ABB RobotStudio station: 码垛.rspag

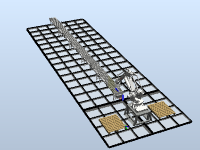
--- station ---
Station PartC (saved by RobotStudio 6.8.8148.134)
Controller System1, task T_ROB1: task frame (RAPID world) sits at (-2000, 0, 800) mm in the station
Controller System1
  mechanical unit ROB_1: IRB660_180_315__01, 6 joints, base frame (0, 0, 0) mm
Layout (positions relative to the parent item):
  - 部件_2 [part] at (0, 0, 23.06) mm
  - ChuanSongDai [smart component]
      signals: DO jiance, DO daowei
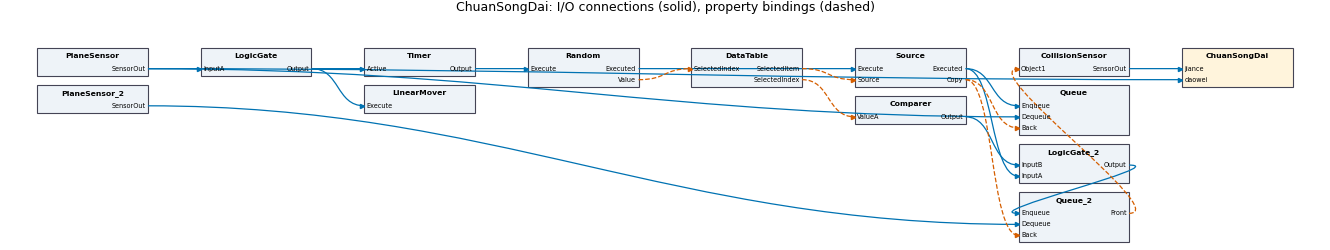
      connections:
        Timer.Output -> Random.Execute
        Random.Executed -> Source.Execute
        LogicGate.Output -> LinearMover.Execute
        Source.Executed -> Queue.Enqueue
        PlaneSensor.SensorOut -> Queue.Dequeue
        LogicGate.Output -> Timer.Active
        Comparer.Output -> LogicGate_2.InputB
        Source.Executed -> LogicGate_2.InputA
        PlaneSensor.SensorOut -> LogicGate.InputA
        LogicGate_2.Output -> Queue_2.Enqueue
        PlaneSensor_2.SensorOut -> Queue_2.Dequeue
        CollisionSensor.SensorOut -> ChuanSongDai.jiance
        PlaneSensor.SensorOut -> ChuanSongDai.daowei
        Random.Value => DataTable.SelectedIndex
        DataTable.SelectedItem => Source.Source
        Source.Copy => Queue.Back
        DataTable.SelectedIndex => Comparer.ValueA
        Source.Copy => Queue_2.Back
        Queue_2.Front => CollisionSensor.Object1
    - Timer [smart component, from Components\Timer.rslib]
        properties: StartTime=0.1; Interval=2.1; Repeat=true; CurrentTime=65.88
    - Random [smart component, from Components\Random.rslib]
        properties: Value=0.822097293018409; Min=0; Max=1
    - DataTable [smart component, from Components\DataTable.rslib]
        properties: DataType=Object; NumItems=2; SelectedIndex=1; SelectedItem=绿; Item0=红; Item1=绿
    - Source [smart component, from Components\Source.rslib]
        properties: Source=绿; Copy=(none); Parent=(none); Position=[12.3 0.05 0.8]; Orientation=[0 0 0]; Transient=false; PhysicsBehavior=0
    - Queue [smart component, from Components\Queue.rslib]
        properties: Back=(none); Front=(none); Queue={f225a319-0da6-49b0-b8ed-6a01384f5e4a};{a5013529-57de-4880-b6b7-02fcb26c5601};{ef2480c9-5506-4bd8-9223-d6bf2a21d1ab};{0e0a0a7f-5876-4dd6-bb12-e12ef663cda4};{136b776b-8417-404b-a9ca-a707fcf896fa};{cb7463a0-53d0-4ea9-9850-c55b52504a23};{429f5040-d4eb-4fed-af85-08b79dd3797b};{eae50fed-bce9-4253-838e-1ef2825aae45};{02ee2a03-807e-4b62-b245-e530b87cc1ef};{56b14a6d-97e9-4dc3-87d2-51b8ae3edd15};{4860391a-c953-42ac-88c5-ff0e025b596f};{e91e6b01-9356-4c41-92bb-629052fa1d8e};{204cb33b-3ecf-4ce5-996c-fe7c59920a57};{7c8b56eb-ca14-4c06-a856-6019091091a4};{df6cc59b-68ab-44d0-93b8-b393a520ffed};{0df2fced-d373-4a8c-8570-b0d5d7a52f36};{2e525211-6f58-4c05-9e0c-770fe7f0b080};{2d23c5ff-243a-4a38-8aa8-df9699042488};{c13a5a0e-5a8c-4728-abd8-7e4e8a2dcb0f};{516486e3-0f15-4dc5-a66e-dbea303b17aa};{aaca48b5-e3d4-4e57-b6f3-5a542b0a9696};{807b33c7-9c87-478a-ab71-3c40786a7147};{5f0bf4f3-3df5-4e69-bf08-9b9bc90daa45};{4c77b5d5-784e-45a8-9efe-70001206c053};{c7fe08fd-9e7d-46e3-a402-e1c13f8510d7};{9c7207f7-ca42-4ffb-ba10-967dca55547d};{a7cd077e-332a-445c-8b65-e16c12a6adc8};{2053ef60-9d1c-42bc-a075-6101035489ef};{a5b924c0-e777-4755-b462-75c4f45590d4};{88fdcb66-1964-4a9a-9fd3-ca14f0fdc147};{ef60cde5-ce41-4944-b10e-df7ae6d2f20b};{427c14b4-609a-4b20-a2be-5ba79a59d804};{fb550f5b-ebcd-4dd1-8fa9-009c54dba658};{c15f4878-baa5-4e14-8903-3b1b5c857eef};{6ededeb0-61e9-45d7-b110-e43846e68698};{d93d9120-f688-4177-bbd5-c04ba3deb883};{aed52de2-8a50-4a30-962b-f942badb32ba};{0d4db61c-ee27-4f7b-9537-b14f67708c8e};{f394902b-ba95-4894-9040-dd871542cf1b};{d8c25479-f3b6-4551-bfd2-063a150a2d78};{38238fd8-de79-4013-ad54-694b5345ed3f};{5bd13c71-3d62-4c6d-bbbc-cc516422125c};{07b92203-4d3e-45b5-80a9-1ec55a767f10};{a74c1ad0-5c37-4e0d-81f5-31d5f0e208c7};{758074db-41a4-4db3-98d0-906284b01602};{6d04588b-afa6-4a99-82e4-be17e8210f91};{348561f2-af5d-4f36-8eda-e8a6df29ee32};{b923b243-db1b-4daf-bb9b-77d6146748ea};{a27ccf1c-a8f2-4afc-910f-c603e908e337};{821874ad-1724-42f4-bffa-9c6221594dbd};{ef4ad952-7e1f-4f76-99cc-78a6cae096f3};{1f82013b-60b1-4451-ab71-6434a119db9b};{6f134922-b885-41ab-a43e-bbaa37394d8e};{7190a3ba-ed00-41fa-baa9-cd3fce09d1b0};{2d9f646b-25f1-493c-9c88-1cc082209cb0};{1953191b-e8a9-4a7b-8072-886da8d2683f};{e6bacfb4-f14c-4f22-ab39-c3f0abe42d56};{8f446c08-29c5-4440-b72c-75c0776f3732};{2ac58cdd-d2f5-4fc3-992e-0072fed280bc};{aa8b40f0-69ac-4ba4-a17b-86b932449b98};{9f18385d-f857-4cee-ba85-427a449adb07};{50a51e2c-eaa8-4e6c-b4d6-fb4141048cc5};{d0e21a90-9519-43be-867c-222b4f1f38a1};{7b820672-940c-4b0d-92fa-2fe77afa0e85};{c9ad62ae-d9f6-4551-810e-0b3d00224a97};{c4bdeaf5-84be-4565-9116-5f2757d6e74e};{59238313-e22c-43d2-a97a-5d6b7997641f};{2edab753-53a4-48c2-8791-8efd26fc352b};{26800b2b-b13d-4846-b0fd-fb68af482c4b};{f6f03289-8baf-42de-9ffb-846ca9933dae};{1e187082-cda8-4acf-9a05-f0e611de5223};{185980c2-df0e-4768-98ff-8c0ecfa9ede1};{c493306c-ebd5-48b7-94e6-332e50b6f699};{c7ce4e63-1a53-4056-bb2e-8373dea2df1b};{00ae25b9-8afd-4489-9d6e-e100ffd902fb};{a46d434a-4951-431b-bf92-58fad4eae258};{0ac38f34-9f27-4a73-b789-8751a30c78c9};{415bd256-8ea2-40f1-afb7-912d3eb54ad5};{5b8083c6-e57c-4f6b-b63b-b57aa365888c};{33a629bd-e383-481d-ba6f-0150e17603ca};{c31adef7-9013-47b8-8c02-a895f65a4230};{bc88b68d-7d5b-4bfa-85ac-205ac4b92c3f};{d122ac05-f8f7-4393-bed0-9e9b9361324e};{227dc145-5e4e-4412-a5e8-4d724cccd912};{96275f03-4ecc-469c-b843-ec3ce2da747c};{3a609a9e-e66e-4842-80c6-6da2b92c4aab};{36be5265-f703-4688-b700-c963585c6167};{78c7701e-fa20-47d5-ad67-3c0217d249c5};{4e3675bd-98e1-4d49-9126-e21ce655e718};{d18456cf-9ef5-48aa-9364-d375af649ce2};{b12914ea-076e-4431-85c1-3df9dfa51120};{477bcbfa-4fa5-46f0-968d-82c75168f6dd};{06c00f79-e598-488f-ab9b-14e942d20a45};{fa9f11b3-aab2-4e3c-9f67-386e2b048710};{965c1e25-d47d-434e-af53-90d46d55ac75};{4f6779af-fb5c-4c41-8ac5-645e945892b7};{961cba95-9dcf-4a6f-ae69-a71c8ac9bd9b};{c1c4ceb7-0aac-4022-8558-a4c71beaa21c};{0f13d351-420a-472e-9a7e-8c0a797d1716};{805a9eb2-f81c-40c7-8f83-e398ffb0342c}; NumberOfObjects=7
    - 600_guide [part, from Equipment\Conveyor Guide 600.rslib]
    - LinearMover [smart component, from Components\LinearMover.rslib]
        properties: Object=Queue; Direction=[-0.001 0 0]; Speed=0.8; Reference=Global; ReferenceObject=(none)
    - PlaneSensor [smart component, from Components\PlaneSensor.rslib]
        properties: Origin=[0 0 0.8]; Axis1=[0 0.6 0]; Axis2=[0 0.1 0.15]; SensedPart=(none)
      - _sensorPart_ [part]
    - LogicGate [smart component, from Components\LogicGate.rslib]
        properties: Operator=NOT; Delay=0
    - Comparer [smart component, from Components\Comparer.rslib]
        properties: ValueA=1; Operator===; ValueB=0
    - LogicGate_2 [smart component, from Components\LogicGate.rslib]
        properties: Operator=AND; Delay=0
    - Queue_2 [smart component, from Components\Queue.rslib]
        properties: Back=(none); Front=(none); Queue={f72ca3a7-ed19-412f-a648-57eb43a8f19a};{0d191394-6de3-422a-92fa-47054eac63d5};{95f6c7dd-c1c0-4261-85cb-418d534c64aa};{209a704b-017e-4eed-926c-5e79c4908886};{0d8d839c-5b7f-48c1-871d-9d79d5e8a973};{1d3bda1c-354e-4164-852e-5573aebfca0e};{d40879a3-4785-47c6-84ec-f61648f74983};{a7cc7dfc-d99a-413b-9ad3-ab5f673166e2};{438c7bca-c9a8-4b7b-9a0a-5120735f9a42};{f225a319-0da6-49b0-b8ed-6a01384f5e4a};{0e0a0a7f-5876-4dd6-bb12-e12ef663cda4};{136b776b-8417-404b-a9ca-a707fcf896fa};{cb7463a0-53d0-4ea9-9850-c55b52504a23};{429f5040-d4eb-4fed-af85-08b79dd3797b};{7c8b56eb-ca14-4c06-a856-6019091091a4};{0df2fced-d373-4a8c-8570-b0d5d7a52f36};{516486e3-0f15-4dc5-a66e-dbea303b17aa};{aaca48b5-e3d4-4e57-b6f3-5a542b0a9696};{5f0bf4f3-3df5-4e69-bf08-9b9bc90daa45};{4c77b5d5-784e-45a8-9efe-70001206c053};{c7fe08fd-9e7d-46e3-a402-e1c13f8510d7};{9c7207f7-ca42-4ffb-ba10-967dca55547d};{88fdcb66-1964-4a9a-9fd3-ca14f0fdc147};{ef60cde5-ce41-4944-b10e-df7ae6d2f20b};{fb550f5b-ebcd-4dd1-8fa9-009c54dba658};{6ededeb0-61e9-45d7-b110-e43846e68698};{758074db-41a4-4db3-98d0-906284b01602};{6d04588b-afa6-4a99-82e4-be17e8210f91};{348561f2-af5d-4f36-8eda-e8a6df29ee32};{b923b243-db1b-4daf-bb9b-77d6146748ea};{6f134922-b885-41ab-a43e-bbaa37394d8e};{1953191b-e8a9-4a7b-8072-886da8d2683f};{e6bacfb4-f14c-4f22-ab39-c3f0abe42d56};{2ac58cdd-d2f5-4fc3-992e-0072fed280bc};{aa8b40f0-69ac-4ba4-a17b-86b932449b98};{9f18385d-f857-4cee-ba85-427a449adb07};{d0e21a90-9519-43be-867c-222b4f1f38a1};{c9ad62ae-d9f6-4551-810e-0b3d00224a97};{c4bdeaf5-84be-4565-9116-5f2757d6e74e};{2edab753-53a4-48c2-8791-8efd26fc352b};{26800b2b-b13d-4846-b0fd-fb68af482c4b};{1e187082-cda8-4acf-9a05-f0e611de5223};{00ae25b9-8afd-4489-9d6e-e100ffd902fb};{a46d434a-4951-431b-bf92-58fad4eae258};{5b8083c6-e57c-4f6b-b63b-b57aa365888c};{33a629bd-e383-481d-ba6f-0150e17603ca};{c31adef7-9013-47b8-8c02-a895f65a4230};{3a609a9e-e66e-4842-80c6-6da2b92c4aab};{36be5265-f703-4688-b700-c963585c6167};{d18456cf-9ef5-48aa-9364-d375af649ce2};{b12914ea-076e-4431-85c1-3df9dfa51120};{fa9f11b3-aab2-4e3c-9f67-386e2b048710};{965c1e25-d47d-434e-af53-90d46d55ac75};{4f6779af-fb5c-4c41-8ac5-645e945892b7};{961cba95-9dcf-4a6f-ae69-a71c8ac9bd9b}; NumberOfObjects=4
    - CollisionSensor [smart component, from Components\CollisionSensor.rslib]
        properties: Object1=(none); Object2=检测; NearMiss=0; Part1=(none); Part2=(none); CollisionType=0
    - PlaneSensor_2 [smart component, from Components\PlaneSensor.rslib]
        properties: Origin=[0 0.7 0.77]; Axis1=[1 0 0]; Axis2=[0 0 1]; SensedPart=(none)
      - _sensorPart_ [part]
  - 红 [part] at (2300, 50, 800) mm
  - 绿 [part]
  - 检测 [part] at (20, 0, 0) mm
  - DiZuo [part] at (-2000, 0, 800) mm
  - IRB660_180_315__01 [mechanism, from Robots\IRB660_180_315__01.rslib] at (-2000, 0, 800) mm; joint values [0.1259, 0.727, 0.7593, 0.1259] (rad or m)
  - TuoPan_Left [part, from B站\木托.rslib] at (-2900, 1230, 0) mm, rotated rx 90 ry 0 rz 90 deg
  - TuoPan_Right [part, from B站\木托.rslib] at (-2900, -2460, 0) mm, rotated rx 90 ry 0 rz 90 deg
  - XiPan [smart component]
      signals: DI zhuaqu
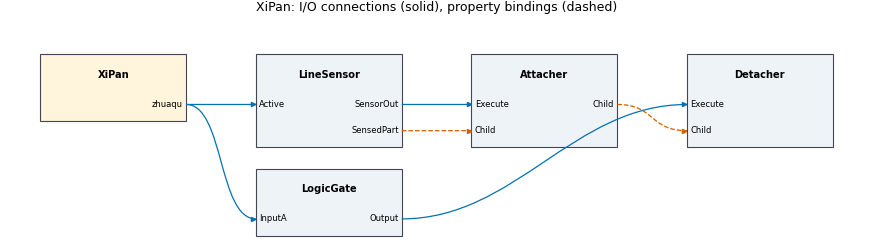
      connections:
        LineSensor.SensorOut -> Attacher.Execute
        LogicGate.Output -> Detacher.Execute
        XiPan.zhuaqu -> LineSensor.Active
        XiPan.zhuaqu -> LogicGate.InputA
        LineSensor.SensedPart => Attacher.Child
        Attacher.Child => Detacher.Child
    - Attacher [smart component, from Components\Attacher.rslib]
        properties: Parent=MyTool; Flange=0; Child=(none); Mount=false; Offset=[0 0 0]; Orientation=[0 0 0]
    - Detacher [smart component, from Components\Detacher.rslib]
        properties: Child=(none); KeepPosition=true
    - LineSensor [smart component, from Components\LineSensor.rslib] at (371, 300, 1200) mm, rotated rx 180 ry 0 rz -180 deg
        properties: Start=[3.44022367537722E-07 -3.10121215152392E-07 -0.0200000204160531]; End=[3.44022367537722E-07 -3.10121215152392E-07 0.029999979583947]; Radius=0.003; SensedPart=(none); SensedPoint=[-1.62997448730469 -2.08514575195312 1.35087182617188]
      - _sensorPart_ [part]
    - MyTool [mechanism] at (371, 300, 1380) mm, rotated rx 180 ry 0 rz -180 deg
        TCP MyTool at (0, 0, 180) mm
        links: 吸盘夹具600_400.
    - LogicGate [smart component, from Components\LogicGate.rslib]
        properties: Operator=NOT; Delay=0
  - 600_guide [part, from Equipment\Conveyor Guide 600.rslib] at (3000, 0, 0) mm
  - 600_guide_2 [part, from Equipment\Conveyor Guide 600.rslib] at (6000, 0, 0) mm
  - 600_guide_3 [part, from Equipment\Conveyor Guide 600.rslib] at (9000, 0, 0) mm
  - 600_guide_4 [part, from Equipment\Conveyor Guide 600.rslib] at (12000, 0, 0) mm
Attachment: LineSensor is attached to MyTool / 吸盘夹具600_400.
Attachment: MyTool is attached to IRB660_180_315__01 / Link6
EventTableEntry 2443: Group=, Trigger=DO_007 2444, Actions=[EventTableActionMechanicalPose 2445], Comment=, ActivationMode=2, Cyclic=false
EventTableTriggerIO 2444: IOValue=[1], IRC5Controller=? -1, Operator=0, SignalSource=? -1
EventTableActionMechanicalPose 2445: VirtualSignal=, Mechanism=? -1, ToPoseName=SyncPosition, VirtualSignalValue=[1]
EventTableEntry 2446: Group=, Trigger=DO_007 2447, Actions=[EventTableActionMechanicalPose 2448], Comment=, ActivationMode=2, Cyclic=false
EventTableTriggerIO 2447: IOValue=[0], IRC5Controller=? -1, Operator=0, SignalSource=? -1
EventTableActionMechanicalPose 2448: VirtualSignal=, Mechanism=? -1, ToPoseName=HomePosition, VirtualSignalValue=[1]
Station logic (signal -> signal, property => property):
  System1.ZhuaQu -> XiPan.zhuaqu
  ChuanSongDai.daowei -> System1.DaoWei
  ChuanSongDai.jiance -> System1.JianCe
Targets, tools, work objects and paths stored in the station and not in the controller backup, written as RAPID:
! task T_ROB1
MODULE CalibData
  PERS tooldata tool1:=[TRUE,[[15.5,0,69.3],[1,0,0,0]],[1,[0,0,1],[1,0,0,0],0,0,0]];
  PERS tooldata tool2:=[TRUE,[[-22.5,0,83.554],[1,0,0,0]],[1,[0,0,1],[1,0,0,0],0,0,0]];
  PERS tooldata tool3:=[TRUE,[[-22.5,0,160.554],[1,0,0,0]],[1,[0,0,1],[1,0,0,0],0,0,0]];
  PERS tooldata Tooldata_4:=[TRUE,[[15.5,0,69.3],[1,0,0,0]],[1,[0,0,1],[1,0,0,0],0,0,0]];
  PERS tooldata Tooldata_5:=[TRUE,[[-22.5,0,83.554],[1,0,0,0]],[1,[0,0,1],[1,0,0,0],0,0,0]];
  PERS tooldata Tooldata_6:=[TRUE,[[-22.5,0,160.554],[1,0,0,0]],[1,[0,0,1],[1,0,0,0],0,0,0]];
ENDMODULE

! task T_ROB1
MODULE Module1
  CONST robtarget Target_10:=[[2810,-1230,2303],[0,0,1,0],[0,0,0,0],[9E+09,9E+09,9E+09,9E+09,9E+09,9E+09]];
ENDMODULE


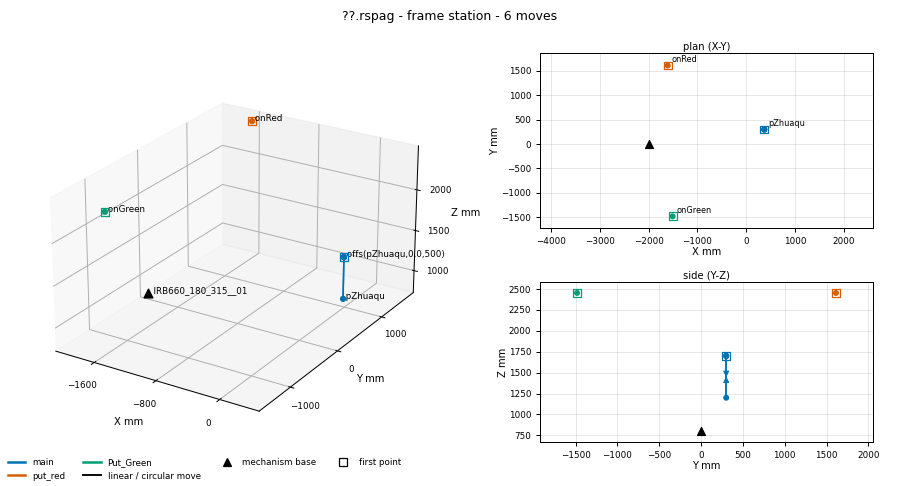
[picture p0: tool path of 码垛.rspag in frame station, 6 of 49 moves have a stored position in this frame; points joined in program order, loops and branches not executed]
--- Backups/System1/RAPID/TASK1/PROGMOD/CalibData.mod ---
MODULE CalibData
	PERS tooldata MyTool:=[TRUE,[[0,0,180],[1,0,0,0]],[1,[0,0,1],[1,0,0,0],0,0,0]];
	TASK PERS wobjdata Work1:=[FALSE,TRUE,"",[[-900,1230,-650],[1,0,0,0]],[[0,0,0],[1,0,0,0]]];
	TASK PERS wobjdata Work2:=[FALSE,TRUE,"",[[620,-1190,-650],[0,0,0,1]],[[0,0,0],[1,0,0,0]]];
ENDMODULE

--- Backups/System1/RAPID/TASK1/PROGMOD/Module1.mod ---
MODULE Module1
	CONST jointtarget Home:=[[0,0,0,0,0,0],[9E+9,9E+9,9E+9,9E+9,9E+9,9E+9]];

	CONST robtarget pZhuaqu:=[[2371.00,300.00,400.00],[1.79568E-6,3.56064E-9,-1,2.27205E-7],[0,0,0,0],[9E+9,9E+9,9E+9,9E+9,9E+9,9E+9]];
	CONST robtarget pFang1:=[[375.00,250.00,400.00],[6.05115E-7,7.10411E-9,1,-1.70585E-6],[1,0,1,0],[9E+9,9E+9,9E+9,9E+9,9E+9,9E+9]];
	CONST robtarget pFang2:=[[1145.00,250.00,400.00],[2.95605E-7,3.17763E-8,-1,1.78569E-6],[0,0,0,0],[9E+9,9E+9,9E+9,9E+9,9E+9,9E+9]];
	CONST robtarget pFang3:=[[250.00,895.00,400.00],[8.4952E-7,0.707106,-0.707107,1.59825E-6],[1,0,0,0],[9E+9,9E+9,9E+9,9E+9,9E+9,9E+9]];
    CONST robtarget pFang4:=[[750.00,895.00,400.00],[8.4952E-7,0.707106,-0.707107,1.59825E-6],[1,0,0,0],[9E+9,9E+9,9E+9,9E+9,9E+9,9E+9]];
	CONST robtarget pFang5:=[[1250.00,895.00,400.00],[8.4952E-7,0.707106,-0.707107,1.59825E-6],[1,0,0,0],[9E+9,9E+9,9E+9,9E+9,9E+9,9E+9]];

    CONST robtarget p2Fang1:=[[250.00,375.00,800.00],[8.4952E-7,0.707106,-0.707107,1.59825E-6],[1,0,0,0],[9E+9,9E+9,9E+9,9E+9,9E+9,9E+9]];
	CONST robtarget p2Fang2:=[[770.00,375.00,800.00],[8.4952E-7,0.707106,-0.707107,1.59825E-6],[1,0,0,0],[9E+9,9E+9,9E+9,9E+9,9E+9,9E+9]];
	CONST robtarget p2Fang3:=[[1250.00,375.00,800.00],[1.27986E-6,-0.707107,-0.707107,-1.27986E-6],[-2,0,0,0],[9E+9,9E+9,9E+9,9E+9,9E+9,9E+9]];
    CONST robtarget p2Fang4:=[[375.00,1020.00,800.00],[6.05115E-7,7.10411E-9,1,-1.70585E-6],[1,0,1,0],[9E+9,9E+9,9E+9,9E+9,9E+9,9E+9]];
    CONST robtarget p2Fang5:=[[1145.00,1020.00,800.00],[6.05115E-7,7.10411E-9,1,-1.70585E-6],[1,0,1,0],[9E+9,9E+9,9E+9,9E+9,9E+9,9E+9]];

    CONST robtarget pPut_green3:=[[250.00,895.00,400.00],[1.03654E-6,0.707107,-0.707107,1.4838E-6],[-1,0,0,0],[9E+9,9E+9,9E+9,9E+9,9E+9,9E+9]];
	CONST robtarget pPut_green1:=[[375.00,250.00,400.00],[1.78435E-6,1,1.03949E-8,3.03588E-7],[-1,0,-1,0],[9E+9,9E+9,9E+9,9E+9,9E+9,9E+9]];
    CONST robtarget pPut_green2:=[[1145.00,250.00,400.00],[1.78435E-6,1,1.03949E-8,3.03588E-7],[-1,0,-1,0],[9E+9,9E+9,9E+9,9E+9,9E+9,9E+9]];
    CONST robtarget pPut_green4:=[[770.00,895.00,400.00],[1.03654E-6,0.707107,-0.707107,1.4838E-6],[-1,0,0,0],[9E+9,9E+9,9E+9,9E+9,9E+9,9E+9]];
    CONST robtarget pPut_green5:=[[1290.00,895.00,400.00],[1.03654E-6,0.707107,-0.707107,1.4838E-6],[-1,0,0,0],[9E+9,9E+9,9E+9,9E+9,9E+9,9E+9]];

    CONST robtarget pPut2_green1:=[[250.00,375.00,800.00],[1.03654E-6,0.707107,-0.707107,1.4838E-6],[-1,0,0,0],[9E+9,9E+9,9E+9,9E+9,9E+9,9E+9]];
    CONST robtarget pPut2_green2:=[[770.00,375.00,800.00],[1.03654E-6,0.707107,-0.707107,1.4838E-6],[-1,0,0,0],[9E+9,9E+9,9E+9,9E+9,9E+9,9E+9]];
    CONST robtarget pPut2_green3:=[[1250.00,375.00,800.00],[1.03654E-6,0.707107,-0.707107,1.4838E-6],[-1,0,0,0],[9E+9,9E+9,9E+9,9E+9,9E+9,9E+9]];
    CONST robtarget pPut2_green4:=[[375.00,1020.00,800.00],[1.78435E-6,1,1.03949E-8,3.03588E-7],[-1,0,-1,0],[9E+9,9E+9,9E+9,9E+9,9E+9,9E+9]];
    CONST robtarget pPut2_green5:=[[1145.00,1020.00,800.00],[1.78435E-6,1,1.03949E-8,3.03588E-7],[-1,0,-1,0],[9E+9,9E+9,9E+9,9E+9,9E+9,9E+9]];

    PERS robtarget put:=[[1250.02,895.106,2000.7],[1.47084E-6,0.707106,-0.707107,1.05485E-6],[0,0,-1,0],[9E+9,9E+9,9E+9,9E+9,9E+9,9E+9]];

    PERS num Layer_red:=6;
    PERS num Layer_green:=6;

    PERS num Number_red:=1;
    PERS num Number_green:=1;

    PERS num Layer1red:=3;
    PERS num Layer2red:=2;
    PERS num Layer1green:=3;
    PERS num Layer2green:=2;

    CONST num long:=750;
    CONST num wide:=500;
    CONST num high:=400;
	CONST robtarget onGreen:=[[129.53,293.34,2303.00],[1.71849E-6,1,-2.69766E-8,5.68225E-7],[-1,0,-1,0],[9E+9,9E+9,9E+9,9E+9,9E+9,9E+9]];
	CONST robtarget onRed:=[[1289.94,382.22,2303.00],[4.41904E-7,0.00933174,-0.999956,1.75522E-6],[0,0,0,0],[9E+9,9E+9,9E+9,9E+9,9E+9,9E+9]];
    !***********************************************************
    !
    ! Module:  Module1
    !
    ! Description:
    !   <Insert description here>
    !
    ! Author: DELL
    !
    ! Version: 1.0
    !
    !***********************************************************


    !***********************************************************
    !
    ! Procedure main
    !
    !   This is the entry point of your program
    !
    !***********************************************************
    PROC main()
        MoveAbsJ Home\NoEOffs,v1000,z50,tool0\WObj:=wobj0;
        Initialize;

        WHILE TRUE DO
        MoveL offs(pZhuaqu,0,0,500),v3000,z50,MyTool\WObj:=wobj0;
        SetDO ZhuaQu,0;
        WaitDI DaoWei,1;
        MoveL pZhuaqu, v1000, fine, MyTool\WObj:=wobj0;
        WaitTime 0.3;
        SetDO ZhuaQu,1;

         IF JianCe=1 and DaoWei=1 THEN
            MoveL offs(pZhuaqu,0,0,500),v3000,z50,MyTool\WObj:=wobj0;
            put_red;
        ELSEIF Jiance=0 and DaoWei=1 THEN
            MoveL offs(pZhuaqu,0,0,500),v3000,z50,MyTool\WObj:=wobj0;
            Put_Green;
        ENDIF

        ENDWHILE
    ENDPROC

    !***********************************************************

    PROC Initialize()

     Layer_red:=1;
     Layer_green:=1;
     Number_red:=1;
     Number_green:=1;

     Layer1red:=0;
     Layer2red:=0;
     Layer1green:=0;
     Layer2green:=0;
    ENDPROC

    !***********************************************************

    PROC put_red()
      IF Layer_red MOD 2=1 THEN

        TEST Number_red
        CASE 1:
        MoveJ offs(pFang1,0,0,Layer1red*800+500),v3000,z50,MyTool\WObj:=Work1;
        MoveJ offs(pFang1,0,0,Layer1red*800),v3000,fine,MyTool\WObj:=Work1;

        CASE 2:
        MoveJ offs(pFang2,0,0,Layer1red*800+500),v3000,z50,MyTool\WObj:=Work1;
        MoveJ offs(pFang2,0,0,Layer1red*800),v3000,fine,MyTool\WObj:=Work1;

        CASE 3:
        MoveJ offs(pFang3,0,0,Layer1red*800+500),v3000,z50,MyTool\WObj:=Work1;
        MoveJ offs(pFang3,0,0,Layer1red*800),v3000,fine,MyTool\WObj:=Work1;

        CASE 4:
        MoveJ offs(pFang4,0,0,Layer1red*800+500),v3000,z50,MyTool\WObj:=Work1;
        MoveJ offs(pFang4,0,0,Layer1red*800),v3000,fine,MyTool\WObj:=Work1;

        CASE 5:
        MoveJ offs(pFang5,0,0,Layer1red*800+500),v3000,z50,MyTool\WObj:=Work1;
        MoveJ offs(pFang5,0,0,Layer1red*800),v3000,fine,MyTool\WObj:=Work1;

        ENDTEST

        IF Number_red=5 THEN
         Layer1red:=Layer1red+1;
        ENDIF

      ENDIF

      IF Layer_red MOD 2=0 THEN
        TEST Number_red
        CASE 1:
        MoveJ offs(p2Fang1,0,0,Layer2red*800+500),v3000,z50,MyTool\WObj:=Work1;
        MoveJ offs(p2Fang1,0,0,Layer2red*800),v3000,fine,MyTool\WObj:=Work1;

        CASE 2:
        MoveJ offs(p2Fang2,0,0,Layer2red*800+500),v3000,z50,MyTool\WObj:=Work1;
        MoveJ offs(p2Fang2,0,0,Layer2red*800),v3000,fine,MyTool\WObj:=Work1;

        CASE 3:
        MoveJ offs(p2Fang3,0,0,Layer2red*800+500),v3000,z50,MyTool\WObj:=Work1;
        MoveJ offs(p2Fang3,0,0,Layer2red*800),v3000,fine,MyTool\WObj:=Work1;

        CASE 4:
        MoveJ offs(p2Fang4,0,0,Layer2red*800+500),v3000,z50,MyTool\WObj:=Work1;
        MoveJ offs(p2Fang4,0,0,Layer2red*800),v3000,fine,MyTool\WObj:=Work1;

        CASE 5:
        MoveJ offs(p2Fang5,0,0,Layer2red*800+500),v3000,z50,MyTool\WObj:=Work1;
        MoveJ offs(p2Fang5,0,0,Layer2red*800),v3000,fine,MyTool\WObj:=Work1;
        ENDTEST

          IF Number_red=5 THEN
           Layer2red:=Layer2red+1;
          ENDIF
       ENDIF

        Reset ZhuaQu;
        Number_red:=Number_red+1;

        IF Number_red>5 THEN
            Number_red:=1;
            Layer_red:=Layer_red+1;
        ENDIF

        put:=CRobT(\Tool:=MyTool\WObj:=Work1);
        MoveJ offs(put,0,0,500),v3000,fine,MyTool\WObj:=Work1;
        MoveJ onRed,v3000,fine,MyTool\WObj:=Work1;
    ENDPROC

    !***********************************************************

        PROC Put_Green()
    IF Layer_green MOD 2=1 THEN

        TEST Number_green
        CASE 1:
        MoveJ offs(pPut_green1,0,0,Layer1green*800+500),v3000,z50,MyTool\WObj:=Work2;
        MoveJ offs(pPut_green1,0,0,Layer1green*800),v3000,fine,MyTool\WObj:=Work2;

        CASE 2:
        MoveJ offs(pPut_green2,0,0,Layer1green*800+500),v3000,z50,MyTool\WObj:=Work2;
        MoveJ offs(pPut_green2,0,0,Layer1green*800),v3000,fine,MyTool\WObj:=Work2;

        CASE 3:
        MoveJ offs(pPut_green3,0,0,Layer1green*800+500),v3000,z50,MyTool\WObj:=Work2;
        MoveJ offs(pPut_green3,0,0,Layer1green*800),v3000,fine,MyTool\WObj:=Work2;

        CASE 4:
        MoveJ offs(pPut_green4,0,0,Layer1green*800+500),v3000,z50,MyTool\WObj:=Work2;
        MoveJ offs(pPut_green4,0,0,Layer1green*800),v3000,fine,MyTool\WObj:=Work2;

        CASE 5:
        MoveJ offs(pPut_green5,0,0,Layer1green*800+500),v3000,z50,MyTool\WObj:=Work2;
        MoveJ offs(pPut_green5,0,0,Layer1green*800),v3000,fine,MyTool\WObj:=Work2;

        ENDTEST

        IF Number_green=5 THEN
         Layer1green:=Layer1green+1;
        ENDIF

    ENDIF

    IF Layer_green MOD 2=0 THEN
        TEST Number_green
        CASE 1:
        MoveJ offs(pPut2_green1,0,0,Layer2green*800+500),v3000,z50,MyTool\WObj:=Work2;
        MoveJ offs(pPut2_green1,0,0,Layer2green*800),v3000,fine,MyTool\WObj:=Work2;

        CASE 2:
        MoveJ offs(pPut2_green2,0,0,Layer2green*800+500),v3000,z50,MyTool\WObj:=Work2;
        MoveJ offs(pPut2_green2,0,0,Layer2green*800),v3000,fine,MyTool\WObj:=Work2;

        CASE 3:
        MoveJ offs(pPut2_green3,0,0,Layer2green*800+500),v3000,z50,MyTool\WObj:=Work2;
        MoveJ offs(pPut2_green3,0,0,Layer2green*800),v3000,fine,MyTool\WObj:=Work2;

        CASE 4:
        MoveJ offs(pPut2_green4,0,0,Layer2green*800+500),v3000,z50,MyTool\WObj:=Work2;
        MoveJ offs(pPut2_green4,0,0,Layer2green*800),v3000,fine,MyTool\WObj:=Work2;

        CASE 5:
        MoveJ offs(pPut2_green5,0,0,Layer2green*800+500),v3000,z50,MyTool\WObj:=Work2;
        MoveJ offs(pPut2_green5,0,0,Layer2green*800),v3000,fine,MyTool\WObj:=Work2;
        ENDTEST

        IF Number_green=5 THEN
         Layer2green:=Layer2green+1;
        ENDIF
    ENDIF

        Reset ZhuaQu;
        Number_green:=Number_green+1;

        IF Number_green>5 THEN
            Number_green:=1;
            Layer_green:=Layer_green+1;
        ENDIF

        put:=CRobT(\Tool:=MyTool\WObj:=Work2);
        MoveJ offs(put,0,0,500),v3000,fine,MyTool\WObj:=Work2;
        MoveJ onGreen,v3000,fine,MyTool\WObj:=Work2;

    ENDPROC

ENDMODULE

--- Backups/System1/SYSPAR/EIO.cfg ---
EIO:CFG_1.0:6:1::
#
EIO_SIGNAL:

      -Name "ZhuaQu" -SignalType "DO"

      -Name "DaoWei" -SignalType "DI"

      -Name "JianCe" -SignalType "DI"
